TYPE InverterCtrl_Typ :
STRUCT
	Start:BOOL;
	ResetError:BOOL;
	SetVelocity:INT;
	ActualVelocity:INT;
END_STRUCT
END_TYPE

(* stored: Version 1.1.0.1, ProductVersion 3.1.4024.3
   DUT InverterCtrl_Typ: Id {14c995cc-eafa-4963-9b3c-5b8a0664c1bc} *)
